Yaskawa INFORM job: R1_W53-A5(180,0)KM-OK_R2.JBI

/JOB
//NAME R1_W53-A5(180,0)KM-OK_R2
///FOLDERNAME KRIS-SCIANA
//POS
///NPOS 88,88,0,5,0,0
///TOOL 0
///POSTYPE PULSE
///PULSE
C00000=6250,-76782,-86706,-6602,54556,71330
///LIMIT ON
C00001=-92663,-139198,-110264,20191,-338,30430
///LIMIT OFF
C00002=-111577,-32962,-81859,22472,97728,49906
C00003=-107780,-69151,-73061,21564,74914,47043
C00004=-108991,-69511,-73240,21928,75160,46643
C00005=-108125,-69258,-73114,21668,74983,46929
C00006=-108125,-69264,-75730,21531,76483,47204
C00007=-117621,-69729,-73984,24277,77870,43984
C00008=-117621,-69493,-70137,24471,75814,43554
C00009=-117621,-69402,-69282,24520,75376,43461
C00010=-117621,-69493,-70137,24471,75814,43554
C00011=-115999,-30718,-51828,23480,83300,45670
C00012=-115999,-31104,-49800,23538,81968,45406
C00013=-115999,-31199,-49180,23559,81572,45328
C00014=-115999,-31104,-49800,23538,81968,45406
C00015=-106921,-26917,-55008,20707,84617,49064
C00016=-107222,-26692,-51834,20853,82965,48677
C00017=-107766,-26892,-51972,21020,83079,48509
C00018=-107222,-26692,-51834,20853,82965,48677
C00019=-104533,-23827,-55295,19924,85724,50052
C00020=-110426,60734,24362,21889,81923,47377
C00021=-110908,60064,26131,22097,80713,46984
C00022=-111296,59897,25939,22206,80843,46866
C00023=-110908,60064,26131,22097,80713,46984
C00024=-110908,60607,23793,22017,82310,47279
C00025=-115927,59000,21966,23435,83913,45819
C00026=-115927,57977,27257,23599,80432,45129
C00027=-115927,57898,28063,23630,79940,45031
C00028=-115927,57977,27257,23599,80432,45129
C00029=-115438,37985,-5121,23224,89196,47018
C00030=-105503,-61482,-91453,20217,88180,50135
C00031=-110518,-95067,-75326,25448,104493,67254
C00032=-109543,-98517,-73266,25325,101434,66951
C00033=-109125,-99754,-72358,25306,100223,66845
C00034=-109125,-98704,-70250,25236,99534,66695
C00035=-109125,-99754,-72358,25306,100223,66845
C00036=-109271,-98731,-72239,25314,100679,66889
C00037=-108845,-102435,-73553,25314,99553,66806
C00038=-109271,-98731,-72239,25314,100679,66889
C00039=-102810,-102082,-74904,21960,97915,67698
C00040=-105287,-102789,-75152,21416,98367,66873
C00041=-102810,-102082,-74904,21960,97915,67698
C00042=-103151,-100933,-75899,21973,99126,67796
C00043=-103951,-97690,-78179,22072,102195,68075
C00044=-107257,-102186,-76413,10931,108592,70034
C00045=-107258,-100380,-72753,10837,107291,69913
C00046=-112980,-104131,-76549,8794,108383,67925
C00047=-107259,-100426,-72861,10839,107332,69917
C00048=-107581,-97187,-70388,10735,107516,69816
C00049=-107118,-100509,-71388,10828,106381,69880
C00050=-108256,-99101,-70337,15518,104986,71666
C00051=-109933,-97756,-65515,33393,95412,78450
C00052=-106611,-96923,-65286,34102,94350,79460
C00053=-105820,-97199,-65380,31409,98835,76028
C00054=-108056,-96592,-65245,24312,106704,68980
C00055=-106650,-96199,-64493,27818,102794,83274
C00056=-107266,-96760,-65778,27977,103379,84733
C00057=-107266,-98376,-68894,28126,104345,84975
C00058=-122843,-113182,-97467,24751,118274,81996
C00059=-129835,-136720,-106856,23968,95426,78599
C00060=-122031,-144606,-118813,21670,55172,80722
C00061=-98554,-52053,-76273,-8136,77037,88849
C00062=-99811,-44360,-64863,-7716,73880,88638
C00063=-100135,-42285,-61231,-8840,68578,88730
C00064=-99407,-48099,-68576,-9102,70170,88862
C00065=-91136,-84120,-86543,-13609,63985,84796
C00066=-92026,-82073,-82060,-13381,62181,84672
C00067=-94422,-69011,-76162,-11907,64826,83469
C00068=-92282,-85842,-88371,-13041,64038,84353
C00069=-96355,-61308,-84875,-4426,92197,81878
C00070=-95984,-62136,-80326,-4483,89018,82107
C00071=-94589,-78161,-87182,-4801,85095,82710
C00072=-94818,-77644,-90492,-4743,87376,82547
C00073=-92917,-101418,-96561,-5233,79041,83514
C00074=-92531,-101358,-95169,-5330,78245,83681
C00075=-90895,-117626,-99808,-5823,72881,84494
C00076=-89952,-135370,-107622,-6185,68664,85042
C00077=-88453,-143067,-104725,-6811,63080,85906
C00078=-87170,-153473,-106248,-7413,58810,86665
C00079=-86786,-160992,-106545,-7816,55198,87069
C00080=-90558,-163951,-107944,-6909,54214,85655
C00081=-122020,-166403,-104868,17331,50735,70544
C00082=-104611,-176380,-105939,3960,44633,78870
C00083=-111868,-169563,-104570,6579,51474,76071
C00084=-139973,-167308,-103995,12166,55330,65477
C00085=-107096,-175612,-110613,4546,48014,77979
C00086=-118025,-149113,-125353,20297,33364,81851
C00087=-16746,-148882,-125293,27639,35588,77892
BC00000=205374,759547,1068166
BC00001=211908,698178,1062837
BC00002=219998,746886,1062839
BC00003=219998,770202,1062839
BC00004=219998,770202,1062839
BC00005=219998,770202,1062839
BC00006=219998,770202,1062839
BC00007=219998,770202,1062839
BC00008=219998,770202,1062839
BC00009=219998,770202,1062839
BC00010=219998,770202,1062839
BC00011=219998,770202,1062839
BC00012=219998,770202,1062839
BC00013=219998,770202,1062839
BC00014=219998,770202,1062839
BC00015=219998,770202,1062839
BC00016=219998,770202,1062839
BC00017=219998,770202,1062839
BC00018=219998,770202,1062839
BC00019=219998,770202,1062839
BC00020=219998,731584,1062839
BC00021=219998,731584,1062839
BC00022=219998,731584,1062839
BC00023=219998,731584,1062839
BC00024=219998,731584,1062839
BC00025=219998,731584,1062839
BC00026=219998,731584,1062839
BC00027=219998,731584,1062839
BC00028=219998,731584,1062839
BC00029=219998,731584,1062839
BC00030=219998,746886,1062839
BC00031=237943,854940,1062845
BC00032=237943,854940,1062845
BC00033=237943,854940,1062845
BC00034=237943,854940,1062845
BC00035=237943,854940,1062845
BC00036=237943,854940,1062845
BC00037=237943,854940,1062845
BC00038=237943,854940,1062845
BC00039=237943,854940,1062845
BC00040=237943,854940,1062845
BC00041=237943,854940,1062845
BC00042=237943,854940,1062845
BC00043=237943,854940,1062845
BC00044=264972,871884,1062845
BC00045=263798,866498,1062845
BC00046=263328,864344,1062845
BC00047=263328,864344,1062845
BC00048=263328,864344,1062845
BC00049=263328,864344,1062845
BC00050=255942,861955,1062845
BC00051=226900,852563,1062845
BC00052=226900,852563,1062845
BC00053=235702,860384,1062845
BC00054=257932,867483,1062841
BC00055=251482,862223,1062845
BC00056=249906,864008,1062845
BC00057=247745,869925,1062845
BC00058=247745,869925,1062845
BC00059=247745,869925,1062845
BC00060=247745,834396,1062845
BC00061=247745,834396,1062845
BC00062=247745,834396,1062845
BC00063=247745,834396,1062845
BC00064=247745,834396,1062845
BC00065=247745,834396,1062845
BC00066=247747,834396,1062843
BC00067=247747,834396,1062843
BC00068=247747,834396,1062843
BC00069=247747,834396,1062843
BC00070=247747,834396,1062841
BC00071=247747,834396,1062841
BC00072=247747,834396,1062841
BC00073=247747,834396,1062841
BC00074=247747,834396,1062841
BC00075=247747,834396,1062841
BC00076=247747,834396,1062841
BC00077=247747,834396,1062841
BC00078=247747,834396,1062841
BC00079=247747,834396,1062841
BC00080=247747,834396,1062841
BC00081=247747,834396,1062841
BC00082=247747,834396,1062841
BC00083=247747,834396,1062841
BC00084=247747,834396,1062841
BC00085=247747,834396,1062841
BC00086=247745,815157,1062845
BC00087=89547,700927,1062845
///POSTYPE BASE
///RECTAN
///RCONF 0,0,0,0,0,0,0,0,0,0,0,0,0,0,0,0,0,0,0,0,0,0,0,0
P00006=0.222,-3.123,-1.508,0.0000,0.0000,0.0000
P00023=0.143,-0.036,0.682,0.0000,0.0000,0.0000
P00025=-2.003,0.006,0.728,0.0000,0.0000,0.0000
P00026=0.562,-0.002,-0.337,0.0000,0.0000,0.0000
P00027=-0.746,0.015,-9.096,0.0000,0.0000,0.0000
//INST
///DATE 2024/07/25 14:02
///ATTR SC,RW
///GROUP1 RB1,BS1
NOP
'r2_W53-A5(180,0)
'Path S1074
MOVJ C00000 BC00000 VJ=20.00
SFTOF
MOVJ C00001 BC00001 VJ=10.00
MOVJ C00002 BC00002 VJ=10.00
MOVJ C00003 BC00003 VJ=10.00
REFP 3 C00004 BC00004
CALL JOB:SEARCH-R1
SET P025 P006
SFTON P025
MOVL C00005 BC00005 V=60.0
MOVL C00006 BC00006 V=100.0
MOVL C00007 BC00007 V=100.0
MOVL C00008 BC00008 V=100.0
REFP 3 C00009 BC00009
CALL JOB:SEARCH-R1
SET P025 P006
SFTON P025
MOVL C00010 BC00010 V=60.0
SFTOF
MOVL C00011 BC00011 V=100.0
MOVL C00012 BC00012 V=100.0
REFP 3 C00013 BC00013
CALL JOB:SEARCH-R1
SET P026 P006
SFTON P026
MOVL C00014 BC00014 V=60.0
MOVL C00015 BC00015 V=100.0
MOVL C00016 BC00016 V=100.0
REFP 3 C00017 BC00017
CALL JOB:SEARCH-R1
SET P026 P006
SFTON P026
MOVL C00018 BC00018 V=60.0
MOVL C00019 BC00019 V=100.0
MOVL C00020 BC00020 V=100.0
MOVL C00021 BC00021 V=100.0
REFP 3 C00022 BC00022
CALL JOB:SEARCH-R1
SET P027 P006
SFTON P027
MOVL C00023 BC00023 V=60.0
MOVL C00024 BC00024 V=100.0
MOVL C00025 BC00025 V=100.0
MOVL C00026 BC00026 V=100.0
REFP 3 C00027 BC00027
CALL JOB:SEARCH-R1
SET P027 P006
SFTON P027
MOVL C00028 BC00028 V=60.0
MOVJ C00029 BC00029 VJ=10.00
MOVJ C00030 BC00030 VJ=10.00
MOVJ C00031 BC00031 VJ=20.00
MOVL C00032 BC00032 V=100.0
MOVL C00033 BC00033 V=60.0
REFP 3 C00034 BC00034
CALL JOB:SEARCH-R1
SET P023 P006
SFTON P023
MOVL C00035 BC00035 V=60.0
MOVL C00036 BC00036 V=60.0
REFP 3 C00037 BC00037
CALL JOB:SEARCH-R1
SET P023 P006
SFTON P023
MOVL C00038 BC00038 V=60.0
MOVL C00039 BC00039 V=60.0
REFP 3 C00040 BC00040
CALL JOB:SEARCH-R1
SET P023 P006
SFTON P023
MOVL C00041 BC00041 V=60.0
MOVL C00042 BC00042 V=100.0
MOVL C00043 BC00043 V=100.0
'Path W1075
SFTOF
MOVJ C00044 BC00044 VJ=20.00
MOVL C00045 BC00045 V=100.0
SFTON P023
MOVL C00046 BC00046 V=100.0 PL=0
REFP 1 C00047 BC00047
REFP 2 C00048 BC00048
MACRO1 MJ#(0) ARGF9
ARCON
MOVL C00049 BC00049 V=10.0
MOVL C00050 BC00050 V=8.3
MOVL C00051 BC00051 V=8.3
MOVL C00052 BC00052 V=8.3
MOVL C00053 BC00053 V=8.3
MOVL C00054 BC00054 V=8.3
MOVL C00055 BC00055 V=8.3
ARCOF
MOVL C00056 BC00056 V=100.0
MOVL C00057 BC00057 V=100.0
MOVJ C00058 BC00058 VJ=20.00
MOVJ C00059 BC00059 VJ=20.00
SFTOF
MOVJ C00060 BC00060 VJ=50.00
MOVJ C00061 BC00061 VJ=50.00
SFTON P027
MACRO1 MJ#(0) ARGF6
MOVJ C00062 BC00062 VJ=15.00
ARCON
MOVL C00063 BC00063 V=13.3
ARCOF
MOVJ C00064 BC00064 VJ=15.00
MOVJ C00065 BC00065 VJ=15.00
MOVJ C00066 BC00066 VJ=15.00
ARCON
MOVL C00067 BC00067 V=13.3
ARCOF
MOVJ C00068 BC00068 VJ=15.00
SFTOF
MOVJ C00069 BC00069 VJ=15.00
SFTON P026
MOVJ C00070 BC00070 VJ=15.00
ARCON
MOVL C00071 BC00071 V=13.3
ARCOF
MOVJ C00072 BC00072 VJ=15.00
MOVJ C00073 BC00073 VJ=15.00
MOVJ C00074 BC00074 VJ=15.00
ARCON
MOVL C00075 BC00075 V=13.3
ARCOF
MOVJ C00076 BC00076 VJ=15.00
SFTOF
SFTON P025
MOVJ C00077 BC00077 VJ=15.00
ARCON
MOVL C00078 BC00078 V=13.3
MOVL C00079 BC00079 V=13.3
ARCOF
MOVJ C00080 BC00080 VJ=15.00
MOVL C00081 BC00081 V=83.3
ARCON
MOVL C00082 BC00082 V=13.3
MOVL C00083 BC00083 V=13.3
MACRO1 MJ#(0) ARGF12
ARCON
WVON WEV#(50)
MOVL C00084 BC00084 V=13.3
ARCOF
WVOF
SFTOF
MOVJ C00085 BC00085 VJ=15.00
MOVJ C00086 BC00086 VJ=20.00
MOVJ C00087 BC00087 VJ=100.00
SFTOF
END
